FUNCTION_BLOCK FB_TcpIpServer EXTENDS FB_EventLogger 
VAR_INPUT
	Enable					: BOOL;//Enable TCP/IP Commnuication
	LocalHost				: T_IPv4Addr := '127.0.0.1';//TCP/IP Socket IP Address
	LocalPort				: UDINT := 1024;//TCP/IP Socket Port
	ReconnectTime			: TIME := T#3S;//Time until reconnection is attempted
	AcceptPollingTime		: TIME := T#100MS;//Send poll time
	RecievePollingTime		: TIME := T#100MS;//Recieve poll Time
	RecieveTimeOut			: TIME := T#3S;// Recieve timeout
	TxData					: ANY;//Raw send data
	RxData					: ANY;//Raw recieve data
	Delimiter				: BYTE := 0;//String data type delimiter in ASCII format
END_VAR                     
VAR_IN_OUT                  
	Control					: ST_System;
END_VAR                     
VAR_OUTPUT                  
	Listening				: BOOL;//Listening for inoming connections
	Accepted				: BOOL;//Socket connection accepted
	SendRecieveRate			: REAL;//Time to send and recieve data over TCP/IP.
END_VAR
VAR
	{attribute 'tc_no_symbol'}   
	_fb_Listen	 			: FB_SocketListen := ( sSrvNetID := '', tTimeout := DEFAULT_ADS_TIMEOUT );//Listener for incoming connection requests from remote clients
	{attribute 'tc_no_symbol'} 
	_fb_SocketClose			: FB_SocketClose := ( sSrvNetID := '', tTimeout := DEFAULT_ADS_TIMEOUT );//Closes an open TCP/IP or UDP socket.
	{attribute 'tc_no_symbol'} 
	_fb_RemoteSocketClose	: FB_SocketClose := ( sSrvNetID := '', tTimeout := DEFAULT_ADS_TIMEOUT );//Closes an open TCP/IP or UDP socket.
	{attribute 'tc_no_symbol'} 
	_fb_SocketAccept		: FB_SocketAccept := ( sSrvNetID := '', tTimeout := DEFAULT_ADS_TIMEOUT );//Accepts remote client connection requests
	{attribute 'tc_no_symbol'} 
	_fb_SocketSend	 		: FB_SocketSend := ( sSrvNetID := '', tTimeout := DEFAULT_ADS_TIMEOUT );//Sends data to a remote client or remote server via the TwinCAT TCP/IP
	{attribute 'tc_no_symbol'} 
	_fb_SocketReceive		: FB_SocketReceive := ( sSrvNetID := '', tTimeout := DEFAULT_ADS_TIMEOUT );//Receives data from a remote client or remote server via the TwinCAT TCP/IP
	{attribute 'tc_no_symbol'} 
	_fb_ConnectTON			: TON;					//Reconnection Timer
	_eStep					: E_ServerSteps;		//Step Engine
	_Listener 				: T_HSOCKET;			//Connection handle of an open socket
	_Alarm					: BOOL;					//Device Alarm
	_Warning				: BOOL;					//Device Warning
	_Message				: BOOL;					//Device Message
	_AlarmNum				: DINT;					//Device Alarm Number
	_WarningNum				: DINT;					//Device Warning Number
	_MessageNum				: DINT;					//Device Message Number
	_Fault					: BOOL;					//Device Fault
	_FaultTimer_ET			: REAL;					//Fault timer elapsed
	_ExtendedErrorCode		: UDINT;				//Extended Error Code
	_RecieveTimeOut			: BOOL;					//No bytes recieved in time error
	_RecieveBufferOverflow	: BOOL;					//No more free read buffer space error
	_r_Trig					: ARRAY[0..9] OF R_TRIG;//Public Rising Edge Triggers
END_VAR                 	
VAR PERSISTENT          	
	_Name					: STRING[15];			//Name for HMI
	_Description			: STRING[40];			//Description for HMI
	_AlarmMute				: BOOL;					//Alarm Mute
	_FaultTimer_PT			: REAL;					//Fault timer preset time
END_VAR

M_AlarmMonitor();
M_WarningMonitor();
M_MessageMonitor();

IF Control.Inputs.AlarmMuteReset THEN _AlarmMute := FALSE; END_IF

CASE _eStep OF

	SERVER_STATE_IDLE:
		IF Enable XOR Listening THEN
			IF Enable THEN
				_fb_ConnectTON( IN := FALSE );
				_eStep := SERVER_STATE_LISTENER_OPEN_START;
			ELSE
				SendRecieveRate := 0;
				_eStep := SERVER_STATE_REMOTE_CLIENTS_CLOSE;
			END_IF
		ELSIF Listening THEN
			_eStep := SERVER_STATE_REMOTE_CLIENTS_COMM;
		END_IF

	SERVER_STATE_LISTENER_OPEN_START:
		_fb_ConnectTON( IN := TRUE, PT := ReconnectTime );
		IF _fb_ConnectTON.Q THEN
		   _fb_ConnectTON( IN := FALSE );
		   _fb_Listen(  bExecute := FALSE  );
		   _fb_Listen(	sLocalHost	:= LocalHost, nLocalPort:= LocalPort, bExecute:= TRUE );
		    _eStep := SERVER_STATE_LISTENER_OPEN_WAIT;
		END_IF

	SERVER_STATE_LISTENER_OPEN_WAIT:
		_fb_Listen( bExecute := FALSE );
		IF NOT _fb_Listen.bBusy THEN
			IF NOT _fb_Listen.bError THEN
				Listening 	:= TRUE;
				_Listener 	:= _fb_Listen.hListener;
				_eStep 	:= SERVER_STATE_IDLE;
			ELSE
				_eStep := SERVER_STATE_ERROR;
			END_IF
		END_IF

	SERVER_STATE_REMOTE_CLIENTS_COMM:
		_eStep := SERVER_STATE_IDLE;
		IF M_RemoteClient(Enable:= TRUE, Listener := _Listener) THEN (*FB_SocketAccept returned error!*)
			_eStep := SERVER_STATE_REMOTE_CLIENTS_CLOSE;
		END_IF	
		
	SERVER_STATE_REMOTE_CLIENTS_CLOSE:
		_eStep := SERVER_STATE_LISTENER_CLOSE_START; (* close listener socket too *)
		IF NOT M_RemoteClient(Enable:= FALSE, Listener := _Listener) AND Accepted THEN
			_eStep := SERVER_STATE_REMOTE_CLIENTS_CLOSE; (* stay here and close all remote clients first *)
		END_IF
	
	SERVER_STATE_LISTENER_CLOSE_START:
		_fb_SocketClose( bExecute := FALSE );
		_fb_SocketClose(	hSocket	:= _Listener,bExecute:= TRUE );
		_eStep := SERVER_STATE_LISTENER_CLOSE_WAIT;

	SERVER_STATE_LISTENER_CLOSE_WAIT:
		_fb_SocketClose( bExecute := FALSE );
		IF NOT _fb_SocketClose.bBusy THEN
			Listening := FALSE;
			MEMSET( ADR(_Listener), 0, SIZEOF(_Listener));
			IF _fb_SocketClose.bError THEN
				_eStep := SERVER_STATE_ERROR;
			ELSE
				_eStep := SERVER_STATE_IDLE;
			END_IF
		END_IF

	SERVER_STATE_ERROR:
		IF Listening THEN
			_eStep := SERVER_STATE_REMOTE_CLIENTS_CLOSE;
		ELSE
			_eStep := SERVER_STATE_IDLE;
		END_IF

END_CASE

{attribute 'monitoring' := 'variable'}
PROPERTY PUBLIC Alarm : Bool
GET
Alarm := _Alarm;
END_GET
END_PROPERTY

{attribute 'monitoring' := 'variable'}
PROPERTY PUBLIC AlarmMute : BOOL
SET
AlarmMute := _AlarmMute;
END_SET
END_PROPERTY

{attribute 'monitoring' := 'variable'}
PROPERTY PUBLIC Description : String[40]
GET
Description := _Description;
END_GET
SET
_Description := Description;
END_SET
END_PROPERTY

{attribute 'monitoring' := 'variable'}
PROPERTY PUBLIC Fault : Bool
SET
_Fault := Fault;
END_SET
END_PROPERTY

{attribute 'monitoring' := 'variable'}
PROPERTY PUBLIC FaultTimer_PT : real
GET
FaultTimer_PT := _FaultTimer_PT;
END_GET
SET
_FaultTimer_PT := FaultTimer_PT;
END_SET
END_PROPERTY

METHOD PRIVATE M_AlarmMonitor
VAR_INPUT
END_VAR
VAR_INST
END_VAR
VAR_INST // added by the converter: edge detectors and wires of the graphical bodies
    _w1, _w2, _w3, _w4, _w5 : BOOL;
    _rt1, _rt2, _rt3, _rt4, _rt5, _rt6, _rt7, _rt8 : R_TRIG;
END_VAR
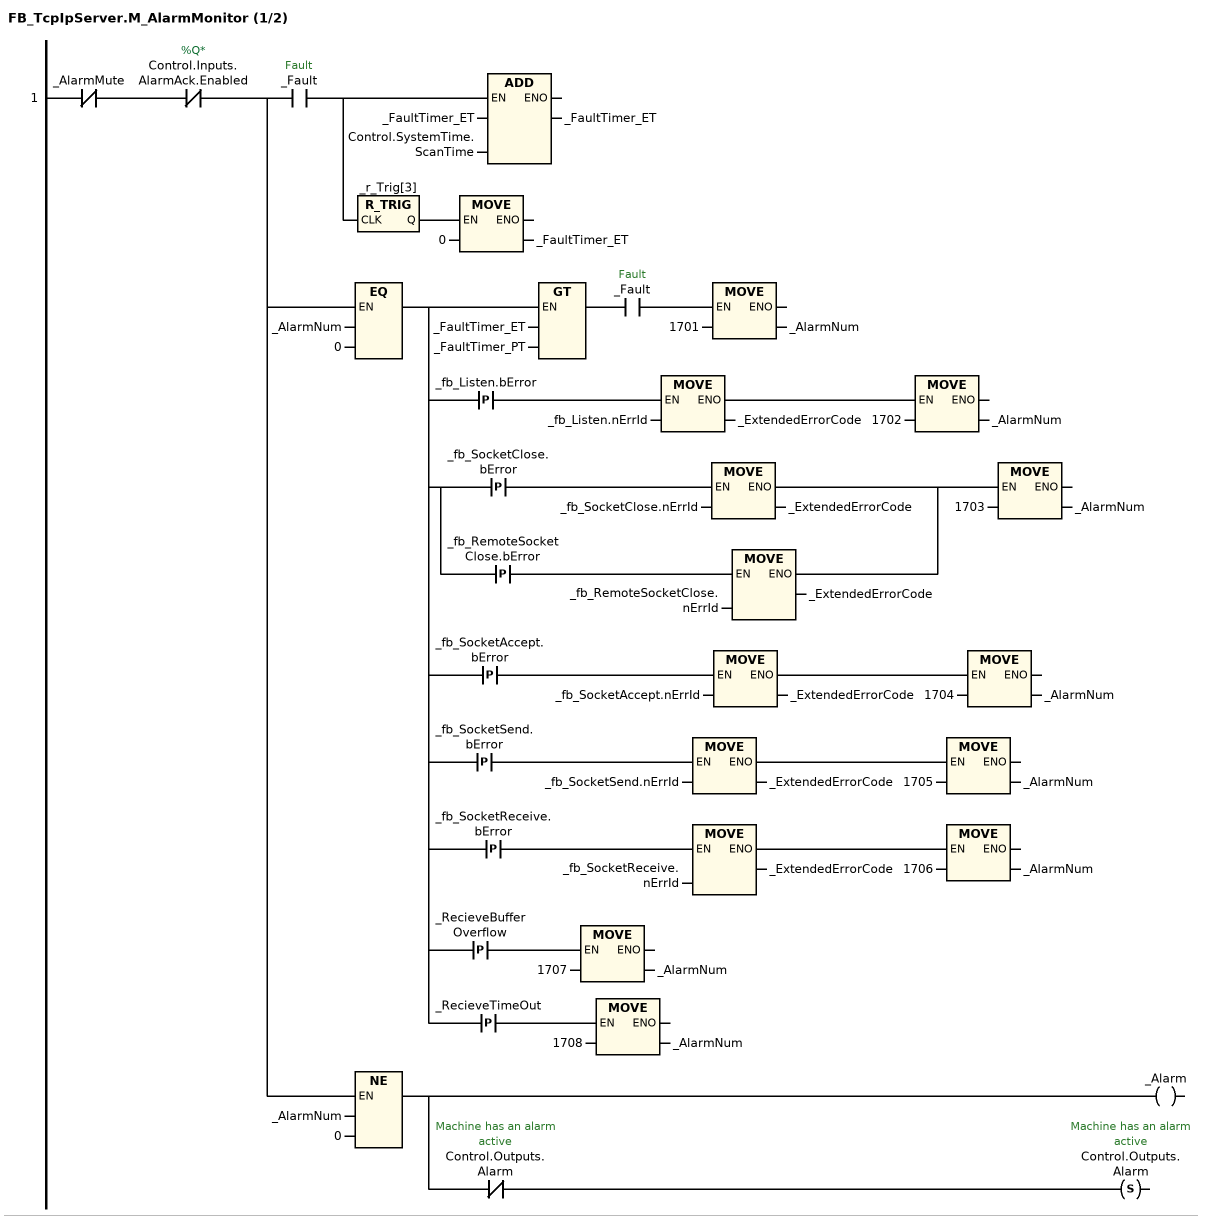
// NETWORK 1
//   Control.Inputs.AlarmAck.Enabled: AT %Q*
//   _Fault: Fault
//   _FaultTimer_ET: Fault timer elapsed
//   Control.SystemTime.ScanTime: Last scan time (Seconds)
//   _FaultTimer_PT: Fault timer preset time
//   Control.Outputs.Alarm: Machine has an alarm active
_w1 := NOT _AlarmMute AND NOT Control.Inputs.AlarmAck.Enabled;
_w2 := _w1 AND _Fault;
IF _w2 THEN _FaultTimer_ET := _FaultTimer_ET + Control.SystemTime.ScanTime; END_IF
_r_Trig[3](CLK := _w2); // R_TRIG
IF _r_Trig[3].Q THEN _FaultTimer_ET := 0; END_IF
_w3 := _w1 AND _AlarmNum = 0;
IF (_w3 AND _FaultTimer_ET > _FaultTimer_PT) AND _Fault THEN _AlarmNum := 1701; END_IF
_rt1(CLK := _fb_Listen.bError);
IF _w3 AND _rt1.Q THEN _ExtendedErrorCode := _fb_Listen.nErrId; END_IF
IF _w3 AND _rt1.Q THEN _AlarmNum := 1702; END_IF
_rt2(CLK := _fb_SocketClose.bError);
IF _w3 AND _rt2.Q THEN _ExtendedErrorCode := _fb_SocketClose.nErrId; END_IF
_rt3(CLK := _fb_RemoteSocketClose.bError);
IF _w3 AND _rt3.Q THEN _ExtendedErrorCode := _fb_RemoteSocketClose.nErrId; END_IF
IF _w3 AND _rt2.Q OR _w3 AND _rt3.Q THEN _AlarmNum := 1703; END_IF
_rt4(CLK := _fb_SocketAccept.bError);
IF _w3 AND _rt4.Q THEN _ExtendedErrorCode := _fb_SocketAccept.nErrId; END_IF
IF _w3 AND _rt4.Q THEN _AlarmNum := 1704; END_IF
_rt5(CLK := _fb_SocketSend.bError);
IF _w3 AND _rt5.Q THEN _ExtendedErrorCode := _fb_SocketSend.nErrId; END_IF
IF _w3 AND _rt5.Q THEN _AlarmNum := 1705; END_IF
_rt6(CLK := _fb_SocketReceive.bError);
IF _w3 AND _rt6.Q THEN _ExtendedErrorCode := _fb_SocketReceive.nErrId; END_IF
IF _w3 AND _rt6.Q THEN _AlarmNum := 1706; END_IF
_rt7(CLK := _RecieveBufferOverflow);
IF _w3 AND _rt7.Q THEN _AlarmNum := 1707; END_IF
_rt8(CLK := _RecieveTimeOut);
IF _w3 AND _rt8.Q THEN _AlarmNum := 1708; END_IF
_w4 := _w1 AND _AlarmNum <> 0;
_Alarm := _w4;
Control.Outputs.Alarm S= _w4 AND NOT Control.Outputs.Alarm;

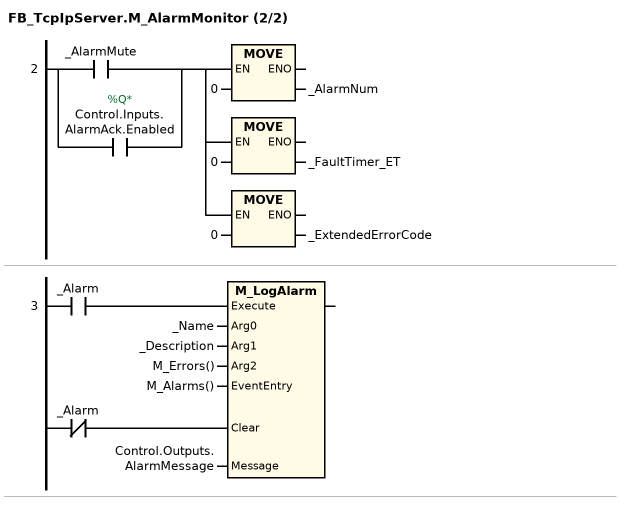
// NETWORK 2
//   Control.Inputs.AlarmAck.Enabled: AT %Q*
//   _FaultTimer_ET: Fault timer elapsed
//   _ExtendedErrorCode: Fault timer elapsed
_w5 := _AlarmMute OR Control.Inputs.AlarmAck.Enabled;
IF _w5 THEN _AlarmNum := 0; END_IF
IF _w5 THEN _FaultTimer_ET := 0; END_IF
IF _w5 THEN _ExtendedErrorCode := 0; END_IF

// NETWORK 3
M_LogAlarm(Execute := _Alarm, Arg0 := _Name, Arg1 := _Description, Arg2 := M_Errors(), EventEntry := M_Alarms(), Clear := NOT _Alarm, Message := Control.Outputs.AlarmMessage);
END_METHOD

METHOD M_Alarms : TcEventEntry
VAR_INPUT
END_VAR
CASE _AlarmNum OF
	1701: M_Alarms:= TC_Events.TcTcpIpServer.A_1701;//General error
	1702: M_Alarms:= TC_Events.TcTcpIpServer.A_1702;//Socket listen error
	1703: M_Alarms:= TC_Events.TcTcpIpServer.A_1703;//Socket close error
	1704: M_Alarms:= TC_Events.TcTcpIpServer.A_1704;//Socket accept error	
	1705: M_Alarms:= TC_Events.TcTcpIpServer.A_1705;//Socket send error	
	1706: M_Alarms:= TC_Events.TcTcpIpServer.A_1706;//Socket recieve error	
	1707: M_Alarms:= TC_Events.TcTcpIpServer.A_1707;//Receive buffer overflow
	1708: M_Alarms:= TC_Events.TcTcpIpServer.A_1708;//Receive timeout error
ELSE
	M_Alarms:= TC_Events.TcTcpIpServer.A_Undefined;
END_CASE
END_METHOD

METHOD PRIVATE M_DataExchange : BOOL;
VAR_INPUT
	Socket				: T_HSOCKET;
	Execute				: BOOL;
END_VAR             	
VAR_INST
	{attribute 'tc_no_symbol'} 
	_Busy				: BOOL;
	{attribute 'tc_no_symbol'} 
	_Error 				: BOOL;
	{attribute 'tc_no_symbol'} 
	_eStep				: E_ServerDataExchangeSteps;
	{attribute 'tc_no_symbol'} 
	_fb_ReceiveTON		: TON;
	{attribute 'tc_no_symbol'} 
	_fb_DisconnectTON 	: TON;
	{attribute 'tc_no_symbol'} 
	_cbFrame			: UDINT;
	{attribute 'tc_no_symbol'} 
	_rxBuffer			: ARRAY[0..255] OF BYTE;
	{attribute 'tc_no_symbol'} 
	_SendRecieveRate	: REAL;
	{attribute 'tc_no_symbol'} 
	_cbReceived, _startPos, _endPos, _idx	: UDINT;
END_VAR
_r_Trig[9]( CLK := Execute );
IF _SendRecieveRate > SendRecieveRate THEN SendRecieveRate :=  _SendRecieveRate; END_IF
_SendRecieveRate := _SendRecieveRate + Control.SystemTime.ScanTime;
CASE _eStep OF

	SERVER_DATAEXCHANGE_STATE_IDLE:
		IF _r_Trig[9].Q THEN
			_SendRecieveRate := 0;
			_Busy 	:= TRUE;
			_Error 	:= FALSE;
			_fb_DisconnectTON( IN := FALSE, PT := T#0MS );(* disable timeout check first *)
			_fb_ReceiveTON( IN := FALSE, PT := T#0MS ); (* receive first request immediately *)
			_eStep 	:= SERVER_DATAEXCHANGE_STATE_RECEIVE_START;
		END_IF

	SERVER_DATAEXCHANGE_STATE_RECEIVE_START: (* Receive remote client data *)
		_fb_ReceiveTON(  IN := TRUE );
		IF _fb_ReceiveTON.Q THEN
			_fb_ReceiveTON( IN := FALSE );
			_fb_SocketReceive( bExecute := FALSE );
			MEMSET(ADR( _rxBuffer ),0,SIZEOF( _rxBuffer ));
			IF RxData.TypeClass = DINT_TO_UDINT(IBaseLibrary.TYPE_STRING) THEN
				_fb_SocketReceive( hSocket:= Socket,pDest:= ADR( _rxBuffer ) , cbLen	:= SIZEOF( _rxBuffer ),bExecute	:= TRUE );
			ELSE
				_fb_SocketReceive( hSocket:= Socket,pDest := RxData.pValue, cbLen:=DINT_TO_UDINT(RxData.diSize),bExecute	:= TRUE );
			END_IF
			_eStep := SERVER_DATAEXCHANGE_STATE_RECEIVE_WAIT;
		END_IF

	SERVER_DATAEXCHANGE_STATE_RECEIVE_WAIT:
		_fb_SocketReceive( bExecute := FALSE );
		IF NOT _fb_SocketReceive.bBusy THEN
			IF NOT _fb_SocketReceive.bError THEN

				IF (_fb_SocketReceive.nRecBytes > 0) THEN(* bytes received *)

					IF RxData.TypeClass = DINT_TO_UDINT(IBaseLibrary.TYPE_STRING) THEN
						_startPos 	:= _cbReceived;(* rxBuffer array index of first data byte *)
						_endPos  	:= _cbReceived + _fb_SocketReceive.nRecBytes  - 1;(* rxBuffer array index of last data byte *)
						_cbReceived 	:= _cbReceived + _fb_SocketReceive.nRecBytes;(* calculate the number of received data bytes *)
						_cbFrame	:= 0;(* reset frame length *)
                	
						IF _cbReceived < DINT_TO_UDINT(RxData.diSize) THEN (* no overflow *)
                	
							_fb_ReceiveTON( IN := FALSE, PT := T#0S ); (* bytes received => increase the read (polling) speed *)
							_fb_DisconnectTON( IN := FALSE, PT := RecieveTimeOut);(* bytes received => disable timeout check *)
                	
							(* search for string end delimiter *)
							FOR _idx := _startPos TO _endPos BY 1 DO
								IF _rxBuffer[_idx] = Delimiter THEN(* string end delimiter found *)
									_cbFrame := _idx + 1;(* calculate the length of the received string (inclusive the end delimiter) *)
									MEMCPY(  RxData.pValue, ADR( _rxBuffer ), _cbFrame );(* copy the received string to the output variable (inclusive the end delimiter) *)
									MEMMOVE( ADR( _rxBuffer ), ADR( _rxBuffer[_cbFrame] ),  _cbReceived - _cbFrame  );(* move the reamaining data bytes *)
									_cbReceived := _cbReceived - _cbFrame;(* recalculate the reamaining data byte length *)
									_eStep := SERVER_DATAEXCHANGE_STATE_SEND_START;
									EXIT;
								END_IF
							END_FOR
                	
						ELSE(* there is no more free read buffer space => the answer string should be terminated *)
							_RecieveBufferOverflow := TRUE;
							_eStep := SERVER_DATAEXCHANGE_STATE_ERROR;
						END_IF
					ELSE
						_eStep := SERVER_DATAEXCHANGE_STATE_SEND_START;
					END_IF

				ELSE(* no bytes received *)
					_fb_ReceiveTON( IN := FALSE, PT := RecievePollingTime);(* no bytes received => decrease the read (polling) speed *)
					_fb_DisconnectTON( IN := TRUE, PT := RecieveTimeOut );(* no bytes received => enable timeout check*)
					IF _fb_DisconnectTON.Q THEN (* timeout error*)
						_fb_DisconnectTON( IN := FALSE );
						_RecieveTimeOut:= TRUE;
						_eStep := SERVER_DATAEXCHANGE_STATE_ERROR;
					ELSE(* repeat reading *)
						_eStep := SERVER_DATAEXCHANGE_STATE_RECEIVE_START; (* repeat reading *)
					END_IF
				END_IF
			ELSE(* receive error *)
				_eStep := SERVER_DATAEXCHANGE_STATE_ERROR;
			END_IF
		END_IF

	SERVER_DATAEXCHANGE_STATE_SEND_START:
		_fb_SocketSend( bExecute := FALSE );
		_fb_SocketSend(	hSocket	:= Socket,pSrc	:= TxData.pValue,cbLen	:=DINT_TO_UDINT(TxData.diSize),bExecute:= TRUE );
		_eStep := SERVER_DATAEXCHANGE_STATE_SEND_WAIT;

	SERVER_DATAEXCHANGE_STATE_SEND_WAIT:
		_fb_SocketSend( bExecute := FALSE );
		IF NOT _fb_SocketSend.bBusy THEN
			IF NOT _fb_SocketSend.bError THEN
				_Busy := FALSE;
				_eStep := SERVER_DATAEXCHANGE_STATE_IDLE;
			ELSE
				_eStep := SERVER_DATAEXCHANGE_STATE_ERROR;
			END_IF
		END_IF

	SERVER_DATAEXCHANGE_STATE_ERROR:
		_Busy := FALSE;
		_RecieveTimeOut:= FALSE;
		_RecieveBufferOverflow := FALSE;
		_Error := TRUE;
		_SendRecieveRate := 0;
		_cbReceived := 0;
		_eStep := SERVER_DATAEXCHANGE_STATE_IDLE;
END_CASE

M_DataExchange:= _Busy;
END_METHOD

METHOD PRIVATE M_Errors : STRING(126)
VAR_INPUT
END_VAR
VAR_INST
END_VAR
CASE _ExtendedErrorCode OF	
//Global Error Codes
0	: M_Errors :='';
1	: M_Errors :='1 Internal error';	 	 
2	: M_Errors :='2 No Rtime';	 	 
3	: M_Errors :='3	Allocation locked memory error';	 	 
4	: M_Errors :='4	Insert mailbox error';
5	: M_Errors :='5	Wrong receive HMSG';	 	 
6	: M_Errors :='6	target port not found	ADS Server not started';	 
7	: M_Errors :='7	target machine not found Missing ADS routes';	 
8	: M_Errors :='8	Unknown command ID';	 	 
9	: M_Errors :='9	Bad task ID';	 	 
10	: M_Errors :='10 No IO';	 	 
11	: M_Errors :='11 Unknown ADS command';	 	 
12	: M_Errors :='12 Win 32 error';	 	 
13	: M_Errors :='13 Port not connected';	 	 
14	: M_Errors :='14 Invalid ADS length';	 	 
15	: M_Errors :='15 Invalid AMS Net ID';	 	 
16	: M_Errors :='16 Low Installation level';	 	 
17	: M_Errors :='17 No debug available';	 	 
18	: M_Errors :='18 Port disabled';	 	 
19	: M_Errors :='19 Port already connected';	 	 
20	: M_Errors :='20 ADS Sync Win32 error';	 	 
21	: M_Errors :='21 ADS Sync Timeout';	 	 
22	: M_Errors :='22 ADS Sync AMS error';	 	 
23	: M_Errors :='23 ADS Sync no index map';	 	 
24	: M_Errors :='24 Invalid ADS port';	 	 
25	: M_Errors :='25 No memory';	 	 
26	: M_Errors :='26 TCP send error';	 	 
27	: M_Errors :='27 Host unreachable'; 	 
28	: M_Errors :='28 Invalid AMS fragment';
//Router Error Codes
1280 :	M_Errors :='1280 No locked memory can be allocated'; 
1281 :	M_Errors :='1281 The size of the router memory could not be changed'; 	 
1282 :	M_Errors :='1282 The mailbox has reached the maximum number OF possible messages'; 
1283 :	M_Errors :='1283 The mailbox has reached the maximum number OF possible messages'; 
1284 :	M_Errors :='1284 The port type is unknown'; 	 
1285 :	M_Errors :='1285 Router is not initialised'; 	 
1286 :	M_Errors :='1286 The desired port number is already assigned'; 	 
1287 :	M_Errors :='1287 Port not registered'; 	 
1288 :	M_Errors :='1288 The maximum number of Ports reached'; 	 
1289 :	M_Errors :='1289 The port is invalid'; 	 
1290 :	M_Errors :='1290 TwinCAT Router not active';  
1291 :	M_Errors :='1291 ROUTERERR_FRAGMENTBOXFULL'; 	 	 
1292 :	M_Errors :='1292 ROUTERERR_FRAGMENTTIMEOUT'; 	 	 
1293 :	M_Errors :='1293 ROUTERERR_TOBEREMOVED'; 
//General ADS Error Codes
1792: M_Errors :='1792 error class <device error>';	 	 
1793: M_Errors :='1793 Service is not supported by server';	 	 
1794: M_Errors :='1794 invalid index group';	 	 
1795: M_Errors :='1795 invalid index offset';	 	 
1796: M_Errors :='1796 reading/writing not permitted';	 	 
1797: M_Errors :='1797 parameter size not correct';	 	 
1798: M_Errors :='1798 invalid parameter value(S)';	 	 
1799: M_Errors :='1799 device is not in a ready state';	 	 
1800: M_Errors :='1800 device is busy';	 	 
1801: M_Errors :='1801 invalid context (must be in Windows)';	 	 
1802: M_Errors :='1802 out OF memory';	 	 
1803: M_Errors :='1803 invalid parameter value(s)';	 	 
1804: M_Errors :='1804 not found (files, ...)';	 	 
1805: M_Errors :='1805 syntax error in command or file';	 	 
1806: M_Errors :='1806 objects DO not match';	 	 
1807: M_Errors :='1807 object already exists';	 	 
1808: M_Errors :='1808 symbol not found';	 	 
1809: M_Errors :='1809 symbol version invalid';	
1810: M_Errors :='1810 server is in invalid state';	 	 
1811: M_Errors :='1811 AdsTransMode not supported';	 	 
1812: M_Errors :='1812 notification handle is invalid';	
1813: M_Errors :='1813 notification client not registered';	 	 
1814: M_Errors :='1814 no more notification handles';	 	 
1815: M_Errors :='1815 size for watch too big';	 	 
1816: M_Errors :='1816 device not initialized';	 	 
1817: M_Errors :='1817 device has a timeout';	 	 
1818: M_Errors :='1818 query INTERFACE failed';	 	 
1819: M_Errors :='1819 wrong interface required';	 	 
1820: M_Errors :='1820 class ID is invalid';	 	 
1821: M_Errors :='1821 object ID is invalid';	 	 
1822: M_Errors :='1822 request is pending';	 	 
1823: M_Errors :='1823 request is aborted';	 	 
1824: M_Errors :='1824 signal warning';	 	 
1825: M_Errors :='1825 invalid array index';	 	 
1826: M_Errors :='1826 symbol not active';	
1827: M_Errors :='1827 access denied';	 	 
1828: M_Errors :='1828 missing license';	 	
1836: M_Errors :='1836 exception occured during system start';	
1856: M_Errors :='1856 Error class <client error>';	 	 
1857: M_Errors :='1857 invalid parameter at service';	 	 
1858: M_Errors :='1858 polling list is empty';	 	 
1859: M_Errors :='1859 var connection already in use';	 	 
1860: M_Errors :='1860 invoke ID in use';	 	 
1861: M_Errors :='1861 timeout elapsed'; 	
1862: M_Errors :='1862 error in win32 subsystem';	 	 
1863: M_Errors :='1863 Invalid client timeout value';	 	 
1864: M_Errors :='1864 ads-port not opened';	 	 
1872: M_Errors :='1872 internal error in ads sync';	 	 
1873: M_Errors :='1873 hash table overflow';	 	 
1874: M_Errors :='1874 key not found in hash';	 	 
1875: M_Errors :='1875 no more symbols in cache';	 	 
1876: M_Errors :='1876 invalid response received';	 	 
1877: M_Errors :='1877 sync port is locked';
//RTime Error Codes
4096: M_Errors:= '4096 INTERNAL error in the REAL-TIME system.';
4097: M_Errors:= '4097 Timer value is NOT valid.';
4098: M_Errors:= '4098 Task pointer has the invalid value 0 (zero).';
4099: M_Errors:= '4099 Stack POINTER has the invalid value 0 (zero).';
4100: M_Errors:= '4100 The request task priority is already assigned.';
4101: M_Errors:= '4101 No free TCB (Task Control Block) available. The maximum number OF TCBs is 64.';
4102: M_Errors:= '4102 No free semaphores available. The maximum number of semaphores is 64.';
4103: M_Errors:= '4103 No free space available in the queue. The maximum number OF positions in the queue is 64.';
4109: M_Errors:= '4109 An external synchronization interrupt is already applied.';
4110: M_Errors:= '4110 No external sync interrupt applied.';
4111: M_Errors:= '4111 Application of the external synchronization interrupt has failed.';
4112: M_Errors:= '4112 Call OF a service FUNCTION in the wrong context';
4119: M_Errors:= '4119 Intel VT-x extension is not supported.';
4120: M_Errors:= '4120 Intel VT-x extension is NOT enabled in the BIOS.';
4121: M_Errors:= '4121 Missing function in Intel VT-x extension.';
4122: M_Errors:= '4122 Activation OF Intel VT-x fails.';
//TCP Winsock Error Codes
10060: M_Errors:= '10060 Intel VT-x extension is NOT enabled in the BIOS.';
10061: M_Errors:= '10061 Missing function in Intel VT-x extension.';
10065: M_Errors:= '10065 Activation OF Intel VT-x fails.';
//Internal error codes of the TwinCAT TCP/IP Connection Server
32769: M_Errors:= '32769 No new sockets can be created (for FB_SocketListen AND FB_SocketConnect).';
32770: M_Errors:= '32770 Socket handle is invalid (for FB_SocketReceive, FB_SocketAccept, FB_SocketSend etc.).';
32771: M_Errors:= '32771 Is returned when FB_SocketListen is called, if the TcpIp port listener already exists.';
32772: M_Errors:= '32772 Is returned when FB_SocketReceive is called, if the client socket is no longer connected with the server.';
32773: M_Errors:= '32773 Is returned when FB_SocketAccept is called, if an error was registered in the listener socket.';
//Internal SNMP error codes
36865: M_Errors:= '36865 INCORRECT PARAMETER SIZE';
36866: M_Errors:= '36866 INVALID PARAMETER';
ELSE
	M_Errors := 	CONCAT('Undefined TCP Server Error - ' , TO_STRING( _ExtendedErrorCode));
END_CASE
END_METHOD

METHOD PRIVATE M_MessageMonitor
VAR_INPUT
END_VAR
VAR_INST
END_VAR
VAR_INST // added by the converter: edge detectors and wires of the graphical bodies
    _w1 : BOOL;
    _rt1, _rt2 : R_TRIG;
    _ft1, _ft2 : F_TRIG;
END_VAR
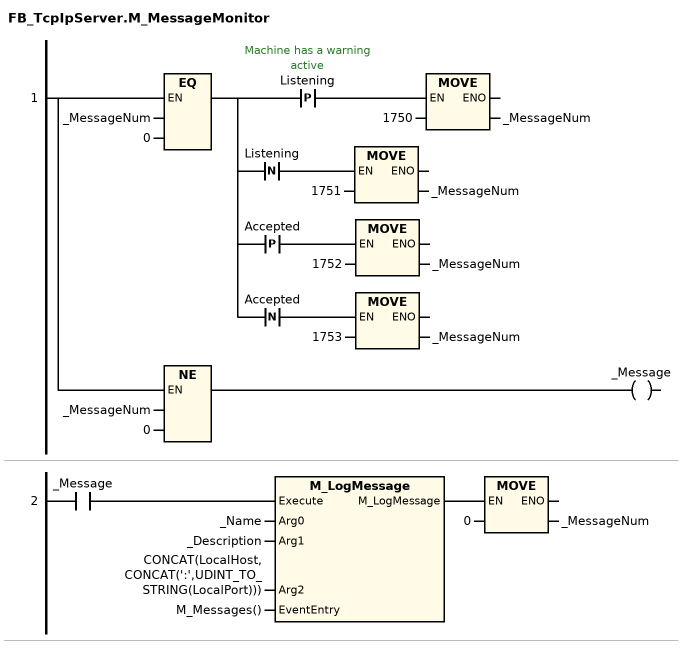
// NETWORK 1
//   Listening: Machine has a warning active
_w1 := _MessageNum = 0;
_rt1(CLK := Listening);
IF _w1 AND _rt1.Q THEN _MessageNum := 1750; END_IF
_ft1(CLK := Listening);
IF _w1 AND _ft1.Q THEN _MessageNum := 1751; END_IF
_rt2(CLK := Accepted);
IF _w1 AND _rt2.Q THEN _MessageNum := 1752; END_IF
_ft2(CLK := Accepted);
IF _w1 AND _ft2.Q THEN _MessageNum := 1753; END_IF
_Message := _MessageNum <> 0;

// NETWORK 2
IF M_LogMessage(Execute := _Message, Arg0 := _Name, Arg1 := _Description, Arg2 := CONCAT(LocalHost,CONCAT(':',UDINT_TO_STRING(LocalPort))), EventEntry := M_Messages()) THEN
    _MessageNum := 0;
END_IF
END_METHOD

METHOD PRIVATE M_Messages : TcEventEntry
VAR_INPUT
END_VAR
CASE _MessageNum OF
	1750: M_Messages:= TC_Events.TcTcpIpServer.M_1750;//Listener socket open
	1751: M_Messages:= TC_Events.TcTcpIpServer.M_1751;//Listener socket closed
	1752: M_Messages:= TC_Events.TcTcpIpServer.M_1752;//Remote client accepted
	1753: M_Messages:= TC_Events.TcTcpIpServer.M_1753;//Remote client closed	
END_CASE
END_METHOD

METHOD PRIVATE M_RemoteClient : BOOL;
VAR_INPUT
	Enable 				: BOOL;
	Listener			: T_HSOCKET;
END_VAR
VAR_INST
	{attribute 'tc_no_symbol'} 
	_Busy				: BOOL;
	{attribute 'tc_no_symbol'} 
	_Error 				: BOOL;
	{attribute 'tc_no_symbol'} 
	_HSocket			: T_HSOCKET;
	{attribute 'tc_no_symbol'} 
	_fb_SocketAcceptTON	: TON;
	{attribute 'tc_no_symbol'} 
	_eStep				: E_ClientSteps;		
END_VAR
CASE _eStep OF

	CLIENT_STATE_IDLE:
		IF Enable XOR Accepted THEN
			_Busy := TRUE;
			_Error := FALSE;
			IF Enable THEN
				_fb_SocketAcceptTON( IN := FALSE );
				_eStep := CLIENT_STATE_CONNECT_START;
			ELSE
				_eStep := CLIENT_STATE_CLOSE_START;
			END_IF
		ELSIF Accepted THEN
			_eStep := CLIENT_STATE_DATAEXCHANGE_START;
		ELSE
			_Busy := FALSE;
		END_IF

	CLIENT_STATE_CONNECT_START:
		_fb_SocketAcceptTON( IN := TRUE, PT := AcceptPollingTime);
		IF _fb_SocketAcceptTON.Q THEN
			_fb_SocketAcceptTON( IN := FALSE );
			_fb_SocketAccept(bExecute := FALSE  );
			_fb_SocketAccept(hListener := Listener,bExecute:= TRUE );
			_eStep := CLIENT_STATE_CONNECT_WAIT;
		END_IF

	CLIENT_STATE_CONNECT_WAIT:
		_fb_SocketAccept( bExecute := FALSE );
		IF NOT _fb_SocketAccept.bBusy THEN
			IF NOT _fb_SocketAccept.bError THEN
				IF _fb_SocketAccept.bAccepted THEN
					Accepted := TRUE;
					_HSocket := _fb_SocketAccept.hSocket;
				END_IF
				_eStep := CLIENT_STATE_IDLE;
			ELSE
				_eStep := CLIENT_STATE_ERROR;
			END_IF
		END_IF

	CLIENT_STATE_DATAEXCHANGE_START:
		M_DataExchange( Execute := FALSE,Socket := _HSocket);
		M_DataExchange( Execute := TRUE ,Socket :=_HSocket);
		_eStep := CLIENT_STATE_DATAEXCHANGE_WAIT;

	CLIENT_STATE_DATAEXCHANGE_WAIT:	
		IF NOT M_DataExchange( Execute := FALSE,Socket := _HSocket) THEN
			_eStep := CLIENT_STATE_IDLE;
		END_IF

	CLIENT_STATE_CLOSE_START:
		_fb_RemoteSocketClose( bExecute := FALSE );
		_fb_RemoteSocketClose(hSocket:= _HSocket,bExecute:= TRUE );
		_eStep := CLIENT_STATE_CLOSE_WAIT;

	CLIENT_STATE_CLOSE_WAIT:
		_fb_RemoteSocketClose( bExecute := FALSE );
		IF NOT _fb_RemoteSocketClose.bBusy THEN
			Accepted := FALSE;
			MEMSET( ADR( _HSocket ),0, SIZEOF( _HSocket ));
			IF _fb_RemoteSocketClose.bError THEN
				_eStep := CLIENT_STATE_ERROR;
			ELSE
				_Busy := FALSE;
				_Error := FALSE;
				_eStep := CLIENT_STATE_IDLE;
			END_IF	
		END_IF

	CLIENT_STATE_ERROR:
		_Error := TRUE;
		IF Accepted THEN
			_eStep := CLIENT_STATE_CLOSE_START;
		ELSE
			_eStep := CLIENT_STATE_IDLE;
			_Busy := FALSE;
		END_IF

END_CASE

M_RemoteClient:= NOT _Busy AND _Error;
END_METHOD

METHOD PRIVATE M_WarningMonitor
VAR_INPUT
END_VAR
VAR_INST
END_VAR
VAR_INST // added by the converter: edge detectors and wires of the graphical bodies
    _w1 : BOOL;
END_VAR
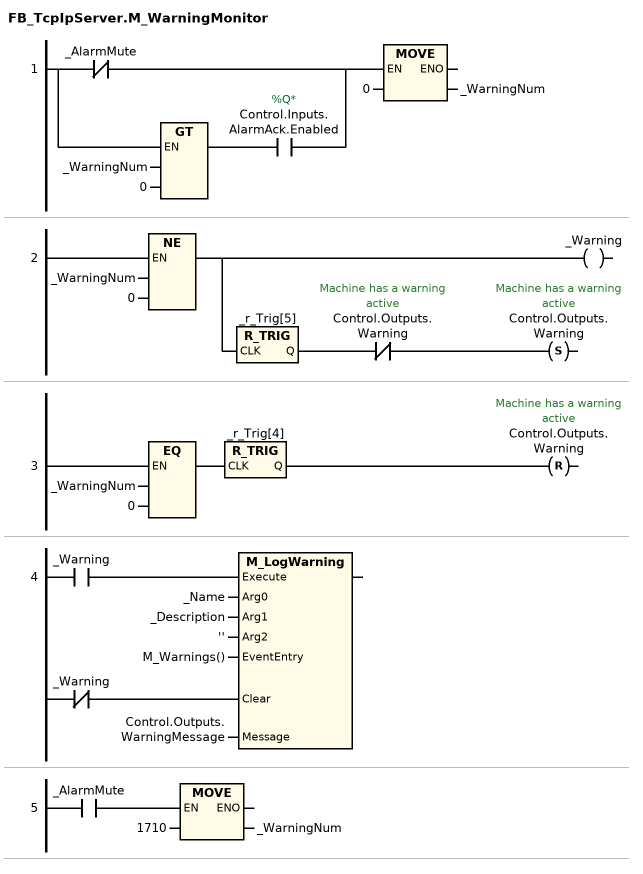
// NETWORK 1
//   Control.Inputs.AlarmAck.Enabled: AT %Q*
IF NOT _AlarmMute OR _WarningNum > 0 AND Control.Inputs.AlarmAck.Enabled THEN _WarningNum := 0; END_IF

// NETWORK 2
//   Control.Outputs.Warning: Machine has a warning active
_w1 := _WarningNum <> 0;
_Warning := _w1;
_r_Trig[5](CLK := _w1); // R_TRIG
Control.Outputs.Warning S= _r_Trig[5].Q AND NOT Control.Outputs.Warning;

// NETWORK 3
//   Control.Outputs.Warning: Machine has a warning active
_r_Trig[4](CLK := _WarningNum = 0); // R_TRIG
Control.Outputs.Warning R= _r_Trig[4].Q;

// NETWORK 4
M_LogWarning(Execute := _Warning, Arg0 := _Name, Arg1 := _Description, Arg2 := '', EventEntry := M_Warnings(), Clear := NOT _Warning, Message := Control.Outputs.WarningMessage);

// NETWORK 5
IF _AlarmMute THEN _WarningNum := 1710; END_IF
END_METHOD

METHOD M_Warnings : TcEventEntry
VAR_INPUT
END_VAR
CASE _WarningNum OF
	1710: M_Warnings:= TC_Events.TcTcpIpServer.W_1710;//Alarm Mute Active				
ELSE
	M_Warnings:=  TC_Events.TcTcpIpServer.W_Undefined;	
END_CASE
END_METHOD

{attribute 'monitoring' := 'variable'}
PROPERTY PUBLIC Name : String[15]
GET
Name := _Name;
END_GET
SET
_Name := Name;
END_SET
END_PROPERTY

{attribute 'monitoring' := 'variable'}
PROPERTY PUBLIC Warning : Bool
GET
Warning := _Warning;
END_GET
END_PROPERTY

END_FUNCTION_BLOCK

(* stored: Version 1.1.0.1, ProductVersion 3.1.4024.3
   POU FB_TcpIpServer: Id {86907fd5-2f80-4033-8615-8b8a40137b8b}, SpecialFunc None
   Property Alarm: Id {756268b0-2ba8-4d96-8e7c-ddb88077d5f1}
   Get Get: Id {8aed1bc3-ad2b-4be8-98a4-f229a097d601}
   Property AlarmMute: Id {54fcffaf-2277-43d8-a673-2d1003164029}
   Set Set: Id {57439e68-8a7e-4fe8-b097-ac759d7d72fb}
   Property Description: Id {5a896fb3-b8e3-4e77-8ded-f8215167d93a}
   Get Get: Id {3c60220a-8dc5-4498-ad9e-e6356be36f74}
   Set Set: Id {1fb7f67c-ec60-4ec6-931c-405ce2f17496}
   Property Fault: Id {8ca0a4ef-1432-4e0b-8024-fc0a401d4a43}
   Set Set: Id {e629d044-7f4b-4628-9792-6c14df63eb15}
   Property FaultTimer_PT: Id {3dfa1591-4055-45fe-9414-f80e1133e6cb}
   Get Get: Id {899d6c50-1241-4929-8c1a-b305eca7007e}
   Set Set: Id {02828da6-8ce8-4dd6-8397-966ed0bda567}
   Method M_AlarmMonitor: Id {9fd6955f-e854-498b-b415-27bf0af0ad93}
   Method M_Alarms: Id {c579e99e-01a7-4595-b5b2-c9c55152cacd}
   Method M_DataExchange: Id {8ab66c67-feda-4c03-8193-c9dafa9c9d7f}
   Method M_Errors: Id {5b63a18b-2e3c-4218-bc03-bf48470c8e98}
   Method M_MessageMonitor: Id {c3784d61-7b15-438c-93f5-00d28054067f}
   Method M_Messages: Id {886b831f-edb7-421d-b6de-82f999b35574}
   Method M_RemoteClient: Id {97c524d2-483f-4c0c-982f-f4a6460377ed}
   Method M_WarningMonitor: Id {54db09ec-04cb-40e9-ab2b-922ec81cad17}
   Method M_Warnings: Id {ed16750a-8bec-4011-8e43-130d8de885f0}
   Property Name: Id {a717dba1-34eb-4356-bb16-5ad1638d79aa}
   Get Get: Id {0d7d6a85-2ee1-4441-8bd7-c8e56561dddf}
   Set Set: Id {aa016fb6-4492-41a9-96ff-7f786c776d79}
   Property Warning: Id {b3f4648b-17e5-454f-a65b-a2d2bd7000c4}
   Get Get: Id {e01eb744-c7cc-4c44-9a35-e24e2f1e7371} *)
